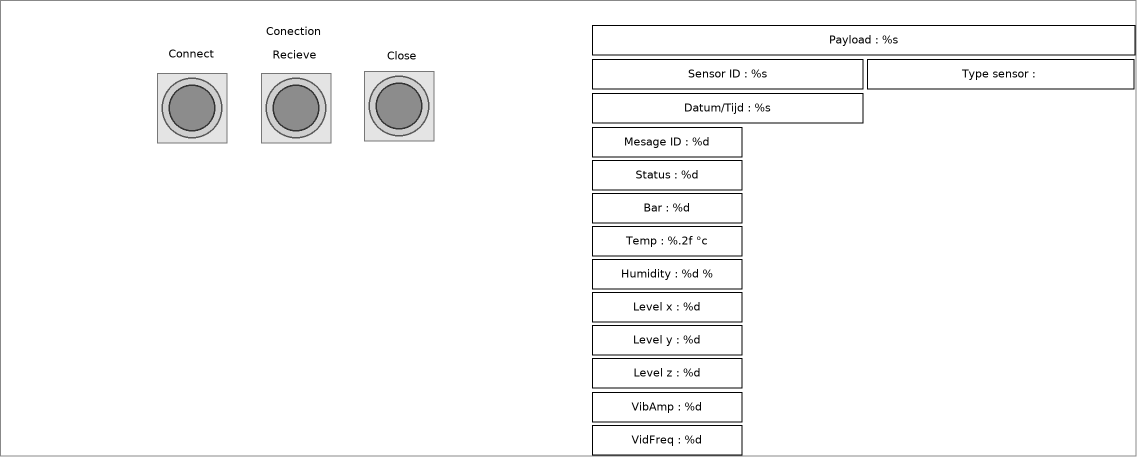
VISUALIZATION Visualization_1  // 1137x457
    PushSwitch (157,73 70x70), variable: Tcp_ip.bConnect, behaviour: TOGGLE, style: Switch-PushSwitch-Gray
    Label (156,39 71x30), "Connect"
    PushSwitch (261,73 70x70), variable: Tcp_ip.bRecieve, behaviour: TOGGLE, style: Switch-PushSwitch-Gray
    Label (261,40 67x30), "Recieve"
    Rectangle (592,25 543x30), "Payload : %s", text variable: PayloadDecoded
    PushSwitch (364,71 70x70), variable: Tcp_ip.FB_close.bExecute, behaviour: TOGGLE, style: Switch-PushSwitch-Gray
    Label (369,41 66x30), "Close"
    Rectangle (592,127 150x30), "Mesage ID : %d", text variable: Decoder.FB_Decoder.MsgID
    Rectangle (592,160 150x30), "Status : %d", text variable: Decoder.Status
    Rectangle (592,193 150x30), "Bar : %d", text variable: Decoder.BaromBar
    Rectangle (592,226 150x30), "Temp : %.2f °c", text variable: Decoder.Temp
    Rectangle (592,259 150x30), "Humidity : %d %", text variable: Decoder.Humidity
    Rectangle (592,292 150x30), "Level x : %d", text variable: Decoder.LevelX
    Rectangle (592,325 150x30), "Level y : %d", text variable: Decoder.LevelY
    Rectangle (592,358 150x30), "Level z : %d", text variable: Decoder.LevelZ
    Rectangle (592,392 150x30), "VibAmp : %d", text variable: Decoder.VibAmp
    Rectangle (592,425 150x30), "VidFreq : %d", text variable: Decoder.VibFreq
    Rectangle (592,59 271x30), "Sensor ID : %s", text variable: Moteeui
    Label (165,17 257x29), "Conection"
    Rectangle (867,59 267x30), "Type sensor :"
    Rectangle (592,93 271x30), "Datum/Tijd : %s", text variable: UserData.Gwrx.TimeRec
END_VISUALIZATION

(* stored: Version 1.1.0.1, ProductVersion 3.1.4022.10
   Visu Visualization_1: Id {1ce6be79-6aa7-4bab-923c-51b6a5c0eb78} *)
